FUNCTION_BLOCK CheckActivePhase (* Basic Function Block Type *)
  (* Standard: 61499-2 *)
  (* Version 0.0, 4/18/2024, SESA371406, Schneider Electric, Template *)
  PACKAGE SE.Nereda;
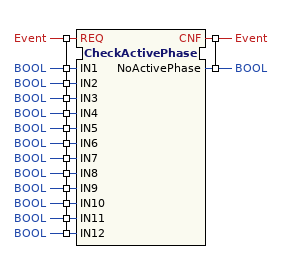
  EVENT_INPUT
    REQ WITH IN1, IN2, IN3, IN4, IN5, IN6, IN7, IN8, IN9, IN10, IN11, IN12; (* Normal Execution Request *)
  END_EVENT
  EVENT_OUTPUT
    CNF WITH NoActivePhase; (* Execution Confirmation *)
  END_EVENT
  VAR_INPUT
    IN1 : BOOL; (* Input event qualifier *)
    IN2 : BOOL;
    IN3 : BOOL;
    IN4 : BOOL;
    IN5 : BOOL;
    IN6 : BOOL;
    IN7 : BOOL;
    IN8 : BOOL;
    IN9 : BOOL;
    IN10 : BOOL;
    IN11 : BOOL;
    IN12 : BOOL;
  END_VAR
  VAR_OUTPUT
    NoActivePhase : BOOL; (* Output event qualifier *)
  END_VAR
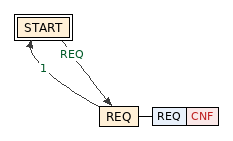
  EC_STATES
    START; (* Initial State *)
    REQ : REQ -> CNF; (* Normal execution *)
  END_STATES
  EC_TRANSITIONS
    REQ TO START := 1;
    START TO REQ := REQ;
  END_TRANSITIONS
  ALGORITHM REQ IN ST: (* Normally executed algorithm *)
;

IF (IN1 = TRUE OR IN2 = TRUE OR IN3 = TRUE) AND
   (IN4 = TRUE OR IN5 = TRUE OR IN6 = TRUE) AND
   (IN7 = TRUE OR IN8 = TRUE OR IN9 = TRUE) AND
   (IN10 = TRUE OR IN11 = TRUE OR IN12 = TRUE) THEN

	NoActivePhase := TRUE;
ELSE
	NoActivePhase := FALSE;
END_IF;
  END_ALGORITHM
  ALGORITHM REQ1 IN ST:
;

NoActivePhase := TRUE;
  END_ALGORITHM
  ALGORITHM REQ2 IN ST:
;
NoActivePhase := FALSE;
  END_ALGORITHM
END_FUNCTION_BLOCK
